// TIA Portal V17 export
// export: Created 2025-03-07T09:18:26.638207Z, ExportSetting WithDefaults, DisplayName Totally Integrated Automation Portal, DisplayVersion V17 Update 8, DisplayName TIA Portal Openness, DisplayVersion V17 Update 8, DisplayName TIA Portal Version Control Interface, DisplayVersion V17, DisplayName SINAMICS Startdrive Advanced, DisplayVersion V17 SP2, DisplayName SINAMICS Startdrive G110M, G120, G120C, G120D, G120P, G115D, DisplayVersion V17 SP2, DisplayName SINAMICS Startdrive G130, G150, S120, S150, SINAMICS MV, S210, DisplayVersion V17 SP2, DisplayName STEP 7 Professional, DisplayVersion V17 Update 8, DisplayName SINUMERIK ONE STEP 7 Toolbox, DisplayVersion V17 Update 12, DisplayName SINUMERIK 840D sl STEP 7 Toolbox, DisplayVersion V17 Update 12, DisplayName STEP 7 Safety, DisplayVersion V17 Update 6, DisplayName WinCC Advanced, DisplayVersion V17 Update 8
FUNCTION "FC1501_MAIN_GAS_VALVE" : Void   // FC1501, LAD
{ S7_Optimized_Access := 'TRUE' }
VERSION : 0.1
// stored: AutoNumber false, IsIECCheckEnabled false, SetENOAutomatically false, UDAEnableTagReadback false
BEGIN

REGION Network 1: CALL FB1405 GENERAL GAS SYSTEM VALVE
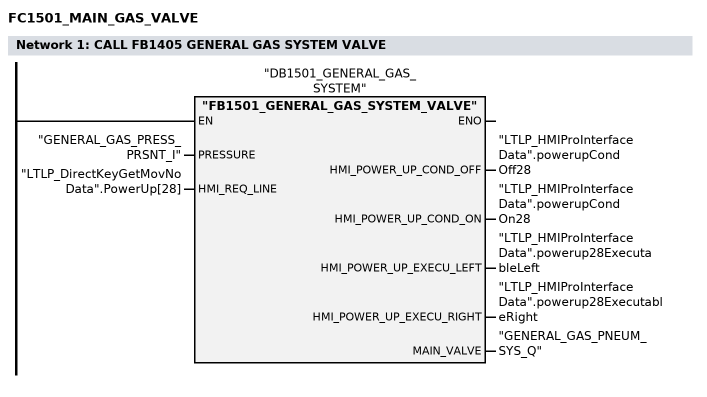
   RUNG wire#powerrail
      "DB1501_GENERAL_GAS_SYSTEM"(PRESSURE := "GENERAL_GAS_PRESS_PRSNT_I", HMI_REQ_LINE := "LTLP_DirectKeyGetMovNoData".PowerUp[28], HMI_POWER_UP_COND_OFF => "LTLP_HMIProInterfaceData".powerupCondOff28, HMI_POWER_UP_COND_ON => "LTLP_HMIProInterfaceData".powerupCondOn28, HMI_POWER_UP_EXECU_LEFT => "LTLP_HMIProInterfaceData".powerup28ExecutableLeft, HMI_POWER_UP_EXECU_RIGHT => "LTLP_HMIProInterfaceData".powerup28ExecutableRight, MAIN_VALVE => "GENERAL_GAS_PNEUM_SYS_Q")
   END_RUNG
   // the same network as SCL:
   "DB1501_GENERAL_GAS_SYSTEM"(PRESSURE := "GENERAL_GAS_PRESS_PRSNT_I",   // "FB1501_GENERAL_GAS_SYSTEM_VALVE"
                           HMI_REQ_LINE := "LTLP_DirectKeyGetMovNoData".PowerUp[28],
                           HMI_POWER_UP_COND_OFF => "LTLP_HMIProInterfaceData".powerupCondOff28,
                           HMI_POWER_UP_COND_ON => "LTLP_HMIProInterfaceData".powerupCondOn28,
                           HMI_POWER_UP_EXECU_LEFT => "LTLP_HMIProInterfaceData".powerup28ExecutableLeft,
                           HMI_POWER_UP_EXECU_RIGHT => "LTLP_HMIProInterfaceData".powerup28ExecutableRight,
                           MAIN_VALVE => "GENERAL_GAS_PNEUM_SYS_Q");
END_REGION
END_FUNCTION
